// TIA Portal V17 export
// export: Created 2025-03-20T13:42:37.7939552Z, ExportSetting WithDefaults, DisplayName Totally Integrated Automation Portal, DisplayVersion V17 Update 8, DisplayName TIA Portal Openness, DisplayVersion V17 Update 8, DisplayName TIA Portal Version Control Interface, DisplayVersion V17, DisplayName SINAMICS Startdrive Advanced, DisplayVersion V17 SP2, DisplayName SINAMICS Startdrive G110M, G120, G120C, G120D, G120P, G115D, DisplayVersion V17 SP2, DisplayName SINAMICS Startdrive G130, G150, S120, S150, SINAMICS MV, S210, DisplayVersion V17 SP2, DisplayName STEP 7 Professional, DisplayVersion V17 Update 8, DisplayName SINUMERIK ONE STEP 7 Toolbox, DisplayVersion V17 Update 12, DisplayName SINUMERIK 840D sl STEP 7 Toolbox, DisplayVersion V17 Update 12, DisplayName STEP 7 Safety, DisplayVersion V17 Update 6, DisplayName WinCC Advanced, DisplayVersion V17 Update 8
FUNCTION "FC2001_FEEDERS_MODES" : Void   // FC2001, LAD
{ S7_Optimized_Access := 'FALSE' }
AUTHOR : ETXETAR
VERSION : 1.0
// stored: AutoNumber false, IsIECCheckEnabled false, SetENOAutomatically false, UDAEnableTagReadback false
   VAR_TEMP
      O_BYTE_0 : Struct   // OPTIONS BYTE 0
         CHANGE_MODE_SEOC_ALARM : Bool;   // CHANGE MODE SEOC ALARM OPTION
         MODE_SELECTED_MEMORY : Bool;   // MODE SELECTED MEMORY OPTION
      END_STRUCT;
   END_VAR
   VAR CONSTANT
      FC_NUMBER : Int := 2021;   // NUMBER
   END_VAR
   VAR_TEMP   // added for the SCL form of the ladder/FBD networks
      _w1 : Bool;
   END_VAR
BEGIN

REGION Network 1: OPTIONS OFF
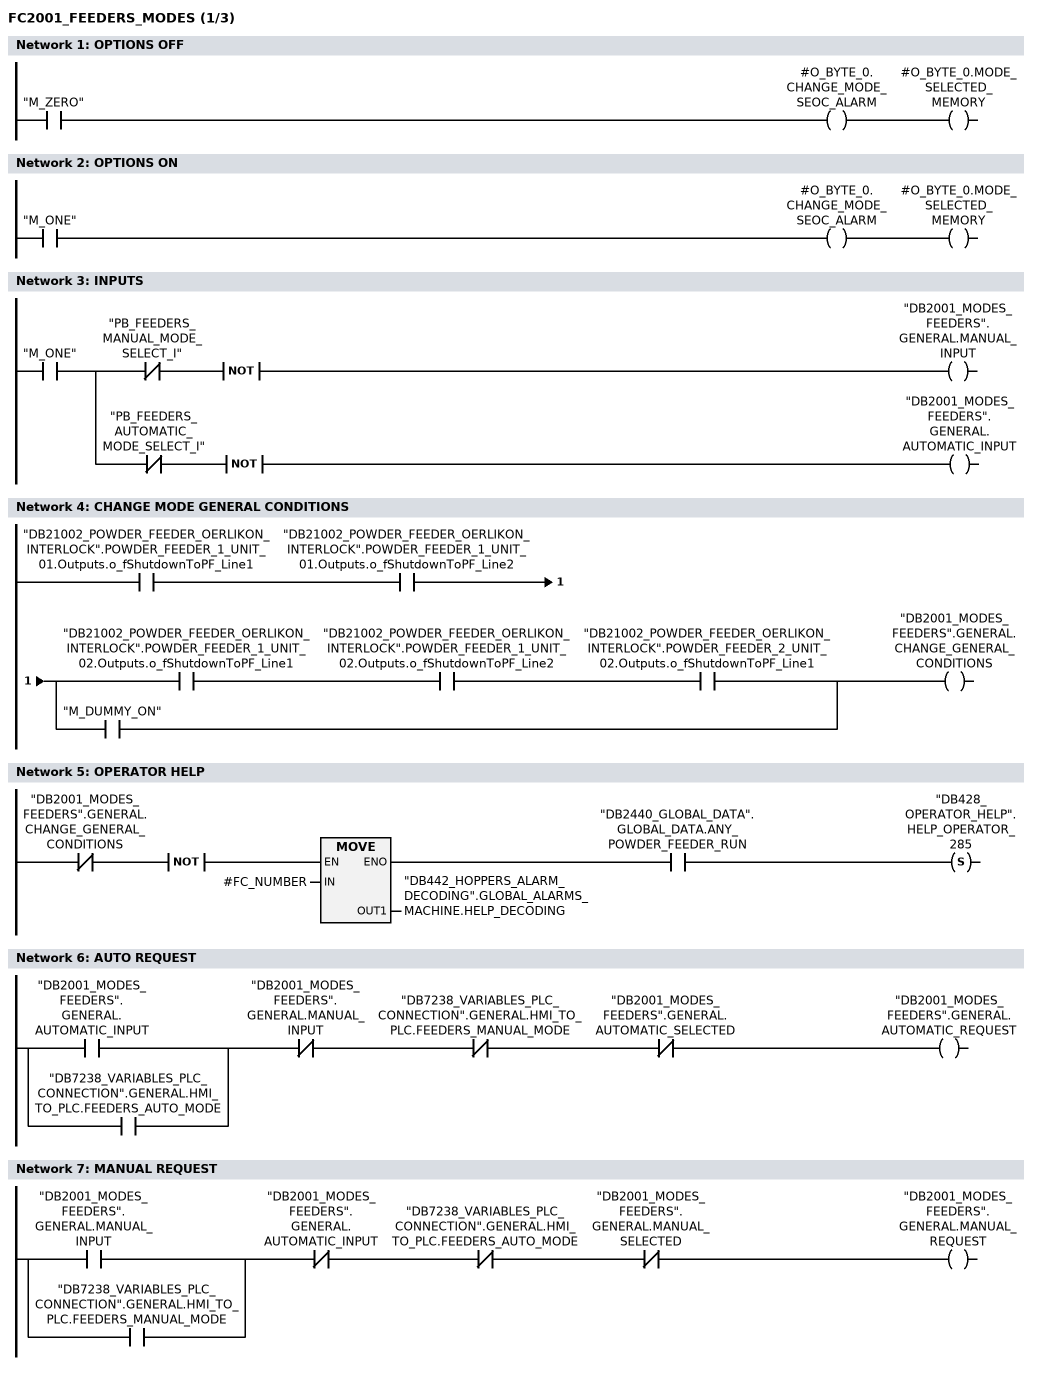
   RUNG wire#powerrail
      Contact( "M_ZERO" )
      Coil( #O_BYTE_0.CHANGE_MODE_SEOC_ALARM )
      Coil( #O_BYTE_0.MODE_SELECTED_MEMORY )
   END_RUNG
   // the same network as SCL:
   #O_BYTE_0.CHANGE_MODE_SEOC_ALARM := "M_ZERO";
   #O_BYTE_0.MODE_SELECTED_MEMORY := "M_ZERO";
END_REGION

REGION Network 2: OPTIONS ON
   RUNG wire#powerrail
      Contact( "M_ONE" )
      Coil( #O_BYTE_0.CHANGE_MODE_SEOC_ALARM )
      Coil( #O_BYTE_0.MODE_SELECTED_MEMORY )
   END_RUNG
   // the same network as SCL:
   #O_BYTE_0.CHANGE_MODE_SEOC_ALARM := "M_ONE";
   #O_BYTE_0.MODE_SELECTED_MEMORY := "M_ONE";
END_REGION

REGION Network 3: INPUTS
   RUNG wire#powerrail
      Contact( "M_ONE" )
      wire#w1
      I_Contact( "PB_FEEDERS_MANUAL_MODE_SELECT_I" )
      Not()
      Coil( "DB2001_MODES_FEEDERS".GENERAL.MANUAL_INPUT )
   END_RUNG
   RUNG wire#w1
      I_Contact( "PB_FEEDERS_AUTOMATIC_MODE_SELECT_I" )
      Not()
      Coil( "DB2001_MODES_FEEDERS".GENERAL.AUTOMATIC_INPUT )
   END_RUNG
   // the same network as SCL:
   "DB2001_MODES_FEEDERS".GENERAL.MANUAL_INPUT := NOT ("M_ONE" AND NOT "PB_FEEDERS_MANUAL_MODE_SELECT_I");
   "DB2001_MODES_FEEDERS".GENERAL.AUTOMATIC_INPUT := NOT ("M_ONE" AND NOT "PB_FEEDERS_AUTOMATIC_MODE_SELECT_I");
END_REGION

REGION Network 4: CHANGE MODE GENERAL CONDITIONS
   RUNG wire#powerrail
      Contact( "DB21002_POWDER_FEEDER_OERLIKON_INTERLOCK".POWDER_FEEDER_1_UNIT_01.Outputs.o_fShutdownToPF_Line1 )
      Contact( "DB21002_POWDER_FEEDER_OERLIKON_INTERLOCK".POWDER_FEEDER_1_UNIT_01.Outputs.o_fShutdownToPF_Line2 )
      wire#w1
      Contact( "DB21002_POWDER_FEEDER_OERLIKON_INTERLOCK".POWDER_FEEDER_1_UNIT_02.Outputs.o_fShutdownToPF_Line1 )
      Contact( "DB21002_POWDER_FEEDER_OERLIKON_INTERLOCK".POWDER_FEEDER_1_UNIT_02.Outputs.o_fShutdownToPF_Line2 )
      Contact( "DB21002_POWDER_FEEDER_OERLIKON_INTERLOCK".POWDER_FEEDER_2_UNIT_02.Outputs.o_fShutdownToPF_Line1 )
      wire#w2
      Coil( "DB2001_MODES_FEEDERS".GENERAL.CHANGE_GENERAL_CONDITIONS )
   END_RUNG
   RUNG wire#w1
      Contact( "M_DUMMY_ON" )
   END_RUNG wire#w2
   // the same network as SCL:
   "DB2001_MODES_FEEDERS".GENERAL.CHANGE_GENERAL_CONDITIONS := "DB21002_POWDER_FEEDER_OERLIKON_INTERLOCK".POWDER_FEEDER_1_UNIT_01.Outputs.o_fShutdownToPF_Line1 AND "DB21002_POWDER_FEEDER_OERLIKON_INTERLOCK".POWDER_FEEDER_1_UNIT_01.Outputs.o_fShutdownToPF_Line2 AND (("DB21002_POWDER_FEEDER_OERLIKON_INTERLOCK".POWDER_FEEDER_1_UNIT_02.Outputs.o_fShutdownToPF_Line1 AND "DB21002_POWDER_FEEDER_OERLIKON_INTERLOCK".POWDER_FEEDER_1_UNIT_02.Outputs.o_fShutdownToPF_Line2 AND "DB21002_POWDER_FEEDER_OERLIKON_INTERLOCK".POWDER_FEEDER_2_UNIT_02.Outputs.o_fShutdownToPF_Line1) OR "M_DUMMY_ON");
END_REGION

REGION Network 5: OPERATOR HELP
   RUNG wire#powerrail
      I_Contact( "DB2001_MODES_FEEDERS".GENERAL.CHANGE_GENERAL_CONDITIONS )
      Not()
      { S7_GenerateENO := "TRUE" } Move(in := #FC_NUMBER, out1 => "DB442_HOPPERS_ALARM_DECODING".GLOBAL_ALARMS_MACHINE.HELP_DECODING)
      Contact( "DB2440_GLOBAL_DATA".GLOBAL_DATA.ANY_POWDER_FEEDER_RUN )
      S_Coil( "DB428_OPERATOR_HELP".HELP_OPERATOR_285 )
   END_RUNG
   // the same network as SCL:
   // ENO of a box is taken as its EN; it also drops when the box reports an error
   #_w1 := NOT (NOT "DB2001_MODES_FEEDERS".GENERAL.CHANGE_GENERAL_CONDITIONS);
   IF #_w1 THEN "DB442_HOPPERS_ALARM_DECODING".GLOBAL_ALARMS_MACHINE.HELP_DECODING := #FC_NUMBER; END_IF;
   IF #_w1 AND "DB2440_GLOBAL_DATA".GLOBAL_DATA.ANY_POWDER_FEEDER_RUN THEN
       "DB428_OPERATOR_HELP".HELP_OPERATOR_285 := TRUE;
   END_IF;
END_REGION

REGION Network 6: AUTO REQUEST
   RUNG wire#powerrail
      Contact( "DB2001_MODES_FEEDERS".GENERAL.AUTOMATIC_INPUT )
      wire#w1
      I_Contact( "DB2001_MODES_FEEDERS".GENERAL.MANUAL_INPUT )
      I_Contact( "DB7238_VARIABLES_PLC_CONNECTION".GENERAL.HMI_TO_PLC.FEEDERS_MANUAL_MODE )
      I_Contact( "DB2001_MODES_FEEDERS".GENERAL.AUTOMATIC_SELECTED )
      Coil( "DB2001_MODES_FEEDERS".GENERAL.AUTOMATIC_REQUEST )
   END_RUNG
   RUNG wire#powerrail
      Contact( "DB7238_VARIABLES_PLC_CONNECTION".GENERAL.HMI_TO_PLC.FEEDERS_AUTO_MODE )
   END_RUNG wire#w1
   // the same network as SCL:
   "DB2001_MODES_FEEDERS".GENERAL.AUTOMATIC_REQUEST := ("DB2001_MODES_FEEDERS".GENERAL.AUTOMATIC_INPUT OR "DB7238_VARIABLES_PLC_CONNECTION".GENERAL.HMI_TO_PLC.FEEDERS_AUTO_MODE) AND NOT "DB2001_MODES_FEEDERS".GENERAL.MANUAL_INPUT AND NOT "DB7238_VARIABLES_PLC_CONNECTION".GENERAL.HMI_TO_PLC.FEEDERS_MANUAL_MODE AND NOT "DB2001_MODES_FEEDERS".GENERAL.AUTOMATIC_SELECTED;
END_REGION

REGION Network 7: MANUAL REQUEST
   RUNG wire#powerrail
      Contact( "DB2001_MODES_FEEDERS".GENERAL.MANUAL_INPUT )
      wire#w1
      I_Contact( "DB2001_MODES_FEEDERS".GENERAL.AUTOMATIC_INPUT )
      I_Contact( "DB7238_VARIABLES_PLC_CONNECTION".GENERAL.HMI_TO_PLC.FEEDERS_AUTO_MODE )
      I_Contact( "DB2001_MODES_FEEDERS".GENERAL.MANUAL_SELECTED )
      Coil( "DB2001_MODES_FEEDERS".GENERAL.MANUAL_REQUEST )
   END_RUNG
   RUNG wire#powerrail
      Contact( "DB7238_VARIABLES_PLC_CONNECTION".GENERAL.HMI_TO_PLC.FEEDERS_MANUAL_MODE )
   END_RUNG wire#w1
   // the same network as SCL:
   "DB2001_MODES_FEEDERS".GENERAL.MANUAL_REQUEST := ("DB2001_MODES_FEEDERS".GENERAL.MANUAL_INPUT OR "DB7238_VARIABLES_PLC_CONNECTION".GENERAL.HMI_TO_PLC.FEEDERS_MANUAL_MODE) AND NOT "DB2001_MODES_FEEDERS".GENERAL.AUTOMATIC_INPUT AND NOT "DB7238_VARIABLES_PLC_CONNECTION".GENERAL.HMI_TO_PLC.FEEDERS_AUTO_MODE AND NOT "DB2001_MODES_FEEDERS".GENERAL.MANUAL_SELECTED;
END_REGION

REGION Network 8: MODE SELECTED MEMORIES
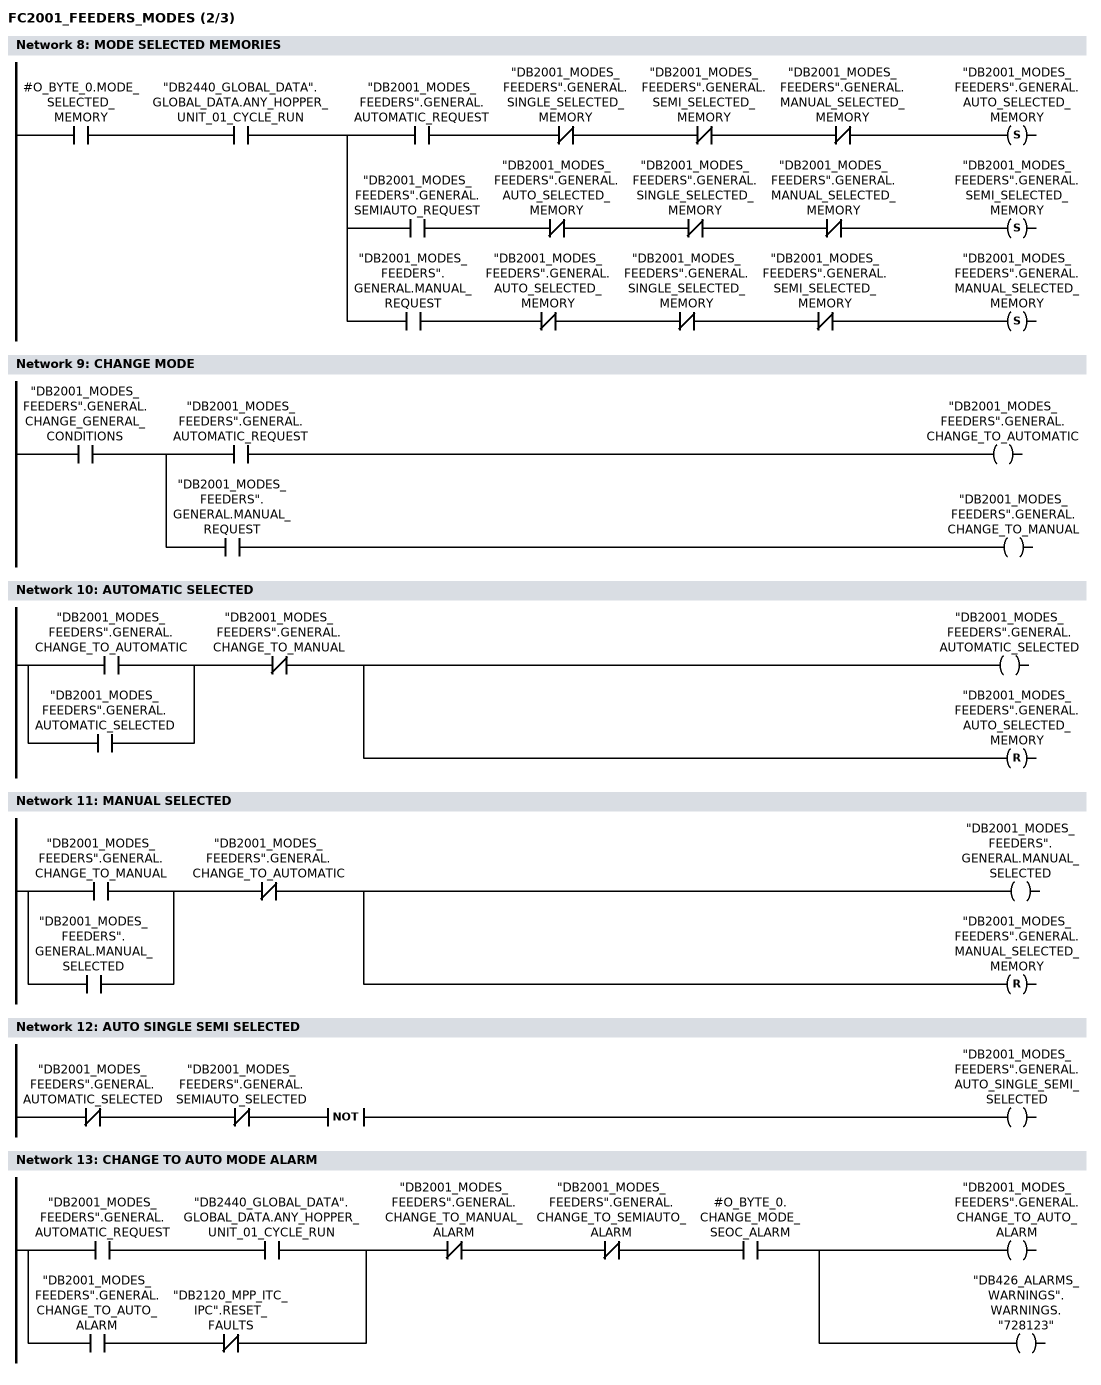
   RUNG wire#powerrail
      Contact( #O_BYTE_0.MODE_SELECTED_MEMORY )
      Contact( "DB2440_GLOBAL_DATA".GLOBAL_DATA.ANY_HOPPER_UNIT_01_CYCLE_RUN )
      wire#w1
      Contact( "DB2001_MODES_FEEDERS".GENERAL.AUTOMATIC_REQUEST )
      I_Contact( "DB2001_MODES_FEEDERS".GENERAL.SINGLE_SELECTED_MEMORY )
      I_Contact( "DB2001_MODES_FEEDERS".GENERAL.SEMI_SELECTED_MEMORY )
      I_Contact( "DB2001_MODES_FEEDERS".GENERAL.MANUAL_SELECTED_MEMORY )
      S_Coil( "DB2001_MODES_FEEDERS".GENERAL.AUTO_SELECTED_MEMORY )
   END_RUNG
   RUNG wire#w1
      Contact( "DB2001_MODES_FEEDERS".GENERAL.SEMIAUTO_REQUEST )
      I_Contact( "DB2001_MODES_FEEDERS".GENERAL.AUTO_SELECTED_MEMORY )
      I_Contact( "DB2001_MODES_FEEDERS".GENERAL.SINGLE_SELECTED_MEMORY )
      I_Contact( "DB2001_MODES_FEEDERS".GENERAL.MANUAL_SELECTED_MEMORY )
      S_Coil( "DB2001_MODES_FEEDERS".GENERAL.SEMI_SELECTED_MEMORY )
   END_RUNG
   RUNG wire#w1
      Contact( "DB2001_MODES_FEEDERS".GENERAL.MANUAL_REQUEST )
      I_Contact( "DB2001_MODES_FEEDERS".GENERAL.AUTO_SELECTED_MEMORY )
      I_Contact( "DB2001_MODES_FEEDERS".GENERAL.SINGLE_SELECTED_MEMORY )
      I_Contact( "DB2001_MODES_FEEDERS".GENERAL.SEMI_SELECTED_MEMORY )
      S_Coil( "DB2001_MODES_FEEDERS".GENERAL.MANUAL_SELECTED_MEMORY )
   END_RUNG
   // the same network as SCL:
   #_w1 := #O_BYTE_0.MODE_SELECTED_MEMORY AND "DB2440_GLOBAL_DATA".GLOBAL_DATA.ANY_HOPPER_UNIT_01_CYCLE_RUN;
   IF #_w1 AND "DB2001_MODES_FEEDERS".GENERAL.AUTOMATIC_REQUEST AND NOT "DB2001_MODES_FEEDERS".GENERAL.SINGLE_SELECTED_MEMORY AND NOT "DB2001_MODES_FEEDERS".GENERAL.SEMI_SELECTED_MEMORY AND NOT "DB2001_MODES_FEEDERS".GENERAL.MANUAL_SELECTED_MEMORY THEN
       "DB2001_MODES_FEEDERS".GENERAL.AUTO_SELECTED_MEMORY := TRUE;
   END_IF;
   IF #_w1 AND "DB2001_MODES_FEEDERS".GENERAL.SEMIAUTO_REQUEST AND NOT "DB2001_MODES_FEEDERS".GENERAL.AUTO_SELECTED_MEMORY AND NOT "DB2001_MODES_FEEDERS".GENERAL.SINGLE_SELECTED_MEMORY AND NOT "DB2001_MODES_FEEDERS".GENERAL.MANUAL_SELECTED_MEMORY THEN
       "DB2001_MODES_FEEDERS".GENERAL.SEMI_SELECTED_MEMORY := TRUE;
   END_IF;
   IF #_w1 AND "DB2001_MODES_FEEDERS".GENERAL.MANUAL_REQUEST AND NOT "DB2001_MODES_FEEDERS".GENERAL.AUTO_SELECTED_MEMORY AND NOT "DB2001_MODES_FEEDERS".GENERAL.SINGLE_SELECTED_MEMORY AND NOT "DB2001_MODES_FEEDERS".GENERAL.SEMI_SELECTED_MEMORY THEN
       "DB2001_MODES_FEEDERS".GENERAL.MANUAL_SELECTED_MEMORY := TRUE;
   END_IF;
END_REGION

REGION Network 9: CHANGE MODE
   RUNG wire#powerrail
      Contact( "DB2001_MODES_FEEDERS".GENERAL.CHANGE_GENERAL_CONDITIONS )
      wire#w1
      Contact( "DB2001_MODES_FEEDERS".GENERAL.AUTOMATIC_REQUEST )
      Coil( "DB2001_MODES_FEEDERS".GENERAL.CHANGE_TO_AUTOMATIC )
   END_RUNG
   RUNG wire#w1
      Contact( "DB2001_MODES_FEEDERS".GENERAL.MANUAL_REQUEST )
      Coil( "DB2001_MODES_FEEDERS".GENERAL.CHANGE_TO_MANUAL )
   END_RUNG
   // the same network as SCL:
   "DB2001_MODES_FEEDERS".GENERAL.CHANGE_TO_AUTOMATIC := "DB2001_MODES_FEEDERS".GENERAL.CHANGE_GENERAL_CONDITIONS AND "DB2001_MODES_FEEDERS".GENERAL.AUTOMATIC_REQUEST;
   "DB2001_MODES_FEEDERS".GENERAL.CHANGE_TO_MANUAL := "DB2001_MODES_FEEDERS".GENERAL.CHANGE_GENERAL_CONDITIONS AND "DB2001_MODES_FEEDERS".GENERAL.MANUAL_REQUEST;
END_REGION

REGION Network 10: AUTOMATIC SELECTED
   RUNG wire#powerrail
      Contact( "DB2001_MODES_FEEDERS".GENERAL.CHANGE_TO_AUTOMATIC )
      wire#w1
      I_Contact( "DB2001_MODES_FEEDERS".GENERAL.CHANGE_TO_MANUAL )
      wire#w2
      Coil( "DB2001_MODES_FEEDERS".GENERAL.AUTOMATIC_SELECTED )
   END_RUNG
   RUNG wire#powerrail
      Contact( "DB2001_MODES_FEEDERS".GENERAL.AUTOMATIC_SELECTED )
   END_RUNG wire#w1
   RUNG wire#w2
      R_Coil( "DB2001_MODES_FEEDERS".GENERAL.AUTO_SELECTED_MEMORY )
   END_RUNG
   // the same network as SCL:
   "DB2001_MODES_FEEDERS".GENERAL.AUTOMATIC_SELECTED := ("DB2001_MODES_FEEDERS".GENERAL.CHANGE_TO_AUTOMATIC OR "DB2001_MODES_FEEDERS".GENERAL.AUTOMATIC_SELECTED) AND NOT "DB2001_MODES_FEEDERS".GENERAL.CHANGE_TO_MANUAL;
   IF "DB2001_MODES_FEEDERS".GENERAL.AUTOMATIC_SELECTED THEN
       "DB2001_MODES_FEEDERS".GENERAL.AUTO_SELECTED_MEMORY := FALSE;
   END_IF;
END_REGION

REGION Network 11: MANUAL SELECTED
   RUNG wire#powerrail
      Contact( "DB2001_MODES_FEEDERS".GENERAL.CHANGE_TO_MANUAL )
      wire#w1
      I_Contact( "DB2001_MODES_FEEDERS".GENERAL.CHANGE_TO_AUTOMATIC )
      wire#w2
      Coil( "DB2001_MODES_FEEDERS".GENERAL.MANUAL_SELECTED )
   END_RUNG
   RUNG wire#powerrail
      Contact( "DB2001_MODES_FEEDERS".GENERAL.MANUAL_SELECTED )
   END_RUNG wire#w1
   RUNG wire#w2
      R_Coil( "DB2001_MODES_FEEDERS".GENERAL.MANUAL_SELECTED_MEMORY )
   END_RUNG
   // the same network as SCL:
   "DB2001_MODES_FEEDERS".GENERAL.MANUAL_SELECTED := ("DB2001_MODES_FEEDERS".GENERAL.CHANGE_TO_MANUAL OR "DB2001_MODES_FEEDERS".GENERAL.MANUAL_SELECTED) AND NOT "DB2001_MODES_FEEDERS".GENERAL.CHANGE_TO_AUTOMATIC;
   IF "DB2001_MODES_FEEDERS".GENERAL.MANUAL_SELECTED THEN
       "DB2001_MODES_FEEDERS".GENERAL.MANUAL_SELECTED_MEMORY := FALSE;
   END_IF;
END_REGION

REGION Network 12: AUTO SINGLE SEMI SELECTED
   RUNG wire#powerrail
      I_Contact( "DB2001_MODES_FEEDERS".GENERAL.AUTOMATIC_SELECTED )
      I_Contact( "DB2001_MODES_FEEDERS".GENERAL.SEMIAUTO_SELECTED )
      Not()
      Coil( "DB2001_MODES_FEEDERS".GENERAL.AUTO_SINGLE_SEMI_SELECTED )
   END_RUNG
   // the same network as SCL:
   "DB2001_MODES_FEEDERS".GENERAL.AUTO_SINGLE_SEMI_SELECTED := NOT (NOT "DB2001_MODES_FEEDERS".GENERAL.AUTOMATIC_SELECTED AND NOT "DB2001_MODES_FEEDERS".GENERAL.SEMIAUTO_SELECTED);
END_REGION

REGION Network 13: CHANGE TO AUTO MODE ALARM
   RUNG wire#powerrail
      Contact( "DB2001_MODES_FEEDERS".GENERAL.AUTOMATIC_REQUEST )
      Contact( "DB2440_GLOBAL_DATA".GLOBAL_DATA.ANY_HOPPER_UNIT_01_CYCLE_RUN )
      wire#w1
      I_Contact( "DB2001_MODES_FEEDERS".GENERAL.CHANGE_TO_MANUAL_ALARM )
      I_Contact( "DB2001_MODES_FEEDERS".GENERAL.CHANGE_TO_SEMIAUTO_ALARM )
      Contact( #O_BYTE_0.CHANGE_MODE_SEOC_ALARM )
      wire#w2
      Coil( "DB2001_MODES_FEEDERS".GENERAL.CHANGE_TO_AUTO_ALARM )
   END_RUNG
   RUNG wire#powerrail
      Contact( "DB2001_MODES_FEEDERS".GENERAL.CHANGE_TO_AUTO_ALARM )
      I_Contact( "DB2120_MPP_ITC_IPC".RESET_FAULTS )
   END_RUNG wire#w1
   RUNG wire#w2
      Coil( "DB426_ALARMS_WARNINGS".WARNINGS."728123" )
   END_RUNG
   // the same network as SCL:
   "DB2001_MODES_FEEDERS".GENERAL.CHANGE_TO_AUTO_ALARM := (("DB2001_MODES_FEEDERS".GENERAL.AUTOMATIC_REQUEST AND "DB2440_GLOBAL_DATA".GLOBAL_DATA.ANY_HOPPER_UNIT_01_CYCLE_RUN) OR ("DB2001_MODES_FEEDERS".GENERAL.CHANGE_TO_AUTO_ALARM AND NOT "DB2120_MPP_ITC_IPC".RESET_FAULTS)) AND NOT "DB2001_MODES_FEEDERS".GENERAL.CHANGE_TO_MANUAL_ALARM AND NOT "DB2001_MODES_FEEDERS".GENERAL.CHANGE_TO_SEMIAUTO_ALARM AND #O_BYTE_0.CHANGE_MODE_SEOC_ALARM;
   "DB426_ALARMS_WARNINGS".WARNINGS."728123" := "DB2001_MODES_FEEDERS".GENERAL.CHANGE_TO_AUTO_ALARM;
END_REGION

REGION Network 14: CHANGE TO MANUAL MODE ALARM
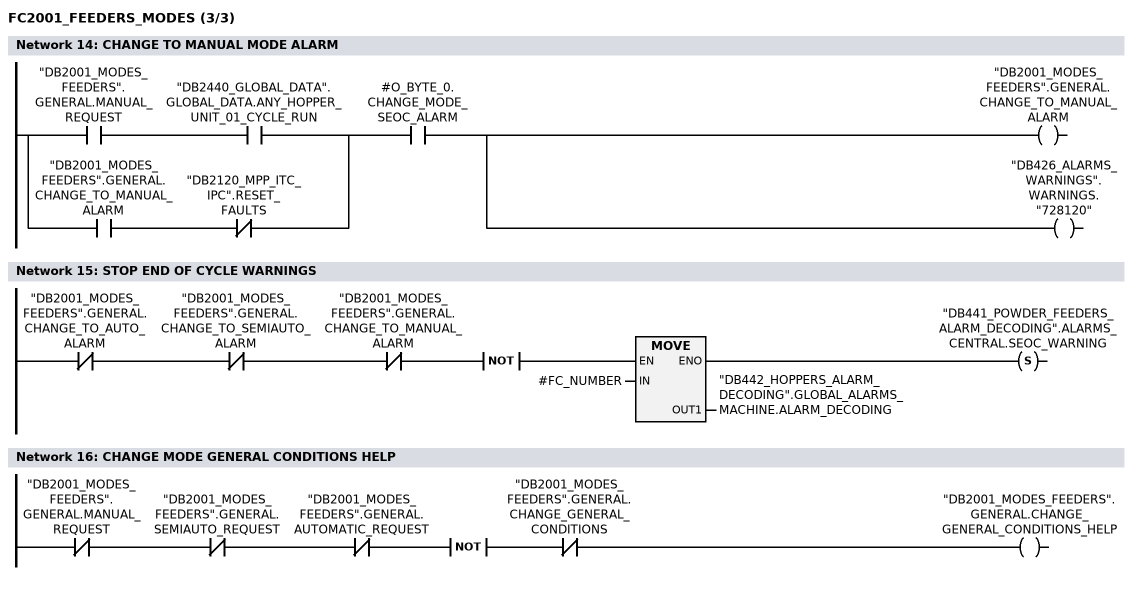
   RUNG wire#powerrail
      Contact( "DB2001_MODES_FEEDERS".GENERAL.MANUAL_REQUEST )
      Contact( "DB2440_GLOBAL_DATA".GLOBAL_DATA.ANY_HOPPER_UNIT_01_CYCLE_RUN )
      wire#w1
      Contact( #O_BYTE_0.CHANGE_MODE_SEOC_ALARM )
      wire#w2
      Coil( "DB2001_MODES_FEEDERS".GENERAL.CHANGE_TO_MANUAL_ALARM )
   END_RUNG
   RUNG wire#powerrail
      Contact( "DB2001_MODES_FEEDERS".GENERAL.CHANGE_TO_MANUAL_ALARM )
      I_Contact( "DB2120_MPP_ITC_IPC".RESET_FAULTS )
   END_RUNG wire#w1
   RUNG wire#w2
      Coil( "DB426_ALARMS_WARNINGS".WARNINGS."728120" )
   END_RUNG
   // the same network as SCL:
   "DB2001_MODES_FEEDERS".GENERAL.CHANGE_TO_MANUAL_ALARM := (("DB2001_MODES_FEEDERS".GENERAL.MANUAL_REQUEST AND "DB2440_GLOBAL_DATA".GLOBAL_DATA.ANY_HOPPER_UNIT_01_CYCLE_RUN) OR ("DB2001_MODES_FEEDERS".GENERAL.CHANGE_TO_MANUAL_ALARM AND NOT "DB2120_MPP_ITC_IPC".RESET_FAULTS)) AND #O_BYTE_0.CHANGE_MODE_SEOC_ALARM;
   "DB426_ALARMS_WARNINGS".WARNINGS."728120" := "DB2001_MODES_FEEDERS".GENERAL.CHANGE_TO_MANUAL_ALARM;
END_REGION

REGION Network 15: STOP END OF CYCLE WARNINGS
   RUNG wire#powerrail
      I_Contact( "DB2001_MODES_FEEDERS".GENERAL.CHANGE_TO_AUTO_ALARM )
      I_Contact( "DB2001_MODES_FEEDERS".GENERAL.CHANGE_TO_SEMIAUTO_ALARM )
      I_Contact( "DB2001_MODES_FEEDERS".GENERAL.CHANGE_TO_MANUAL_ALARM )
      Not()
      { S7_GenerateENO := "TRUE" } Move(in := #FC_NUMBER, out1 => "DB442_HOPPERS_ALARM_DECODING".GLOBAL_ALARMS_MACHINE.ALARM_DECODING)
      S_Coil( "DB441_POWDER_FEEDERS_ALARM_DECODING".ALARMS_CENTRAL.SEOC_WARNING )
   END_RUNG
   // the same network as SCL:
   // ENO of a box is taken as its EN; it also drops when the box reports an error
   IF NOT (NOT "DB2001_MODES_FEEDERS".GENERAL.CHANGE_TO_AUTO_ALARM AND NOT "DB2001_MODES_FEEDERS".GENERAL.CHANGE_TO_SEMIAUTO_ALARM AND NOT "DB2001_MODES_FEEDERS".GENERAL.CHANGE_TO_MANUAL_ALARM) THEN
       "DB442_HOPPERS_ALARM_DECODING".GLOBAL_ALARMS_MACHINE.ALARM_DECODING := #FC_NUMBER;
       "DB441_POWDER_FEEDERS_ALARM_DECODING".ALARMS_CENTRAL.SEOC_WARNING := TRUE;
   END_IF;
END_REGION

REGION Network 16: CHANGE MODE GENERAL CONDITIONS HELP
   RUNG wire#powerrail
      I_Contact( "DB2001_MODES_FEEDERS".GENERAL.MANUAL_REQUEST )
      I_Contact( "DB2001_MODES_FEEDERS".GENERAL.SEMIAUTO_REQUEST )
      I_Contact( "DB2001_MODES_FEEDERS".GENERAL.AUTOMATIC_REQUEST )
      Not()
      I_Contact( "DB2001_MODES_FEEDERS".GENERAL.CHANGE_GENERAL_CONDITIONS )
      Coil( "DB2001_MODES_FEEDERS".GENERAL.CHANGE_GENERAL_CONDITIONS_HELP )
   END_RUNG
   // the same network as SCL:
   "DB2001_MODES_FEEDERS".GENERAL.CHANGE_GENERAL_CONDITIONS_HELP := NOT (NOT "DB2001_MODES_FEEDERS".GENERAL.MANUAL_REQUEST AND NOT "DB2001_MODES_FEEDERS".GENERAL.SEMIAUTO_REQUEST AND NOT "DB2001_MODES_FEEDERS".GENERAL.AUTOMATIC_REQUEST) AND NOT "DB2001_MODES_FEEDERS".GENERAL.CHANGE_GENERAL_CONDITIONS;
END_REGION
END_FUNCTION
